INTERFACE I_CollisionGroup

METHOD AddMoverToThisGroup : HRESULT
VAR_INPUT
	MoverToAdd : I_XtsMover;
END_VAR
END_METHOD

PROPERTY CAGroupXtsIoEnvInterface : I_Mc2CaGroup
GET
END_GET
SET
END_SET
END_PROPERTY

METHOD Disable : BOOL
VAR_INPUT
END_VAR
END_METHOD

METHOD Enable : BOOL
VAR_INPUT
END_VAR
END_METHOD

METHOD GetAxisCount : udint
VAR_INPUT
END_VAR
END_METHOD

PROPERTY GroupRef : reference to AXES_GROUP_REF
GET
END_GET
END_PROPERTY

PROPERTY GroupState : CAGroupStatus
GET
END_GET
END_PROPERTY

METHOD GroupStop : HRESULT
VAR_INPUT
END_VAR
END_METHOD

PROPERTY MyName : string
GET
END_GET
END_PROPERTY

METHOD RemoveAllMovers : HRESULT
VAR_INPUT
END_VAR
END_METHOD

METHOD RemoveAMover : BOOL
VAR_INPUT
	Mover : I_XtsMover;
END_VAR
END_METHOD

METHOD Reset : HRESULT
VAR_INPUT
END_VAR
END_METHOD

END_INTERFACE

(* stored: Version 1.1.0.1
   Itf I_CollisionGroup: Id {3fc566cf-3f15-4187-97a8-f8d156c2ea05}
   Method AddMoverToThisGroup: Id {e0521e35-3414-4dd6-b2e7-4ac92ca8a051}
   Property CAGroupXtsIoEnvInterface: Id {cd5d9462-f9cf-4d35-b22c-6eae8c9cec38}
   Get Get: Id {4b7a5dbd-2b80-4c96-b418-833e5507e708}
   Set Set: Id {a85ceeb9-ae20-4fa6-83c9-e0f32834f786}
   Method Disable: Id {716927af-8c3f-479d-962f-20b060f08214}
   Method Enable: Id {7961c446-8ffb-4a93-bee2-efac793ad03b}
   Method GetAxisCount: Id {c1a4af34-8409-44b5-8d2c-3faa797a2cef}
   Property GroupRef: Id {da70f768-e857-4f18-9014-1c57ab869df0}
   Get Get: Id {ff65d9fd-a0fb-4014-a5bd-11ea974f60f4}
   Property GroupState: Id {ccaa4875-e7b8-4aad-9434-8ae988f5aafa}
   Get Get: Id {6ce504cb-b674-4e50-8b81-3854a9614761}
   Method GroupStop: Id {da0fa42b-dbcd-4e72-85b3-93d42f55308f}
   Property MyName: Id {989d2fa8-4a9f-4077-ad60-57e1e6700080}
   Get Get: Id {962bda42-6307-4da5-99e1-648fbb7790b1}
   Method RemoveAllMovers: Id {ef3d94da-4e03-448c-b177-7286a6d747e3}
   Method RemoveAMover: Id {ef48cf2e-8bac-48d4-bde6-7be9e9dfb88f}
   Method Reset: Id {52cfbceb-29c1-48af-b76e-6022383fab33} *)
